PROGRAM MAIN
VAR
	bInit				: BOOL := TRUE;
	
	fbCell 				: FB_Cell;
	
	fbFiller			: FB_Filler;
	fbCapper			: FB_Capper;
	fbCheckWeigher		: FB_CheckWeigher;
	
	bTest				: ARRAY[0..9] OF BOOL;
	fbSimAxis			: FB_SimAxis;
	fSimTarget			: LREAL := 500;
	fSimVelocity		: LREAL := 100;
END_VAR

// Initialize cell
IF bInit THEN
	fbCell.AddStation(fbFiller);
	fbCell.AddStation(fbCapper);
	fbCell.AddStation(fbCheckWeigher);
	bInit := FALSE;
END_IF

fbCell.Execute();

IF bTest[0] THEN
	IF fbSimAxis.MoveAbsolute(fSimtarget, fSimVelocity) THEN
		bTest[0] := FALSE;
	END_IF
END_IF

END_PROGRAM

(* stored: Version 1.1.0.1, ProductVersion 3.1.4024.12
   POU MAIN: Id {c03723bc-6d53-4d9e-a9ba-46b2795c327c}, SpecialFunc None *)
